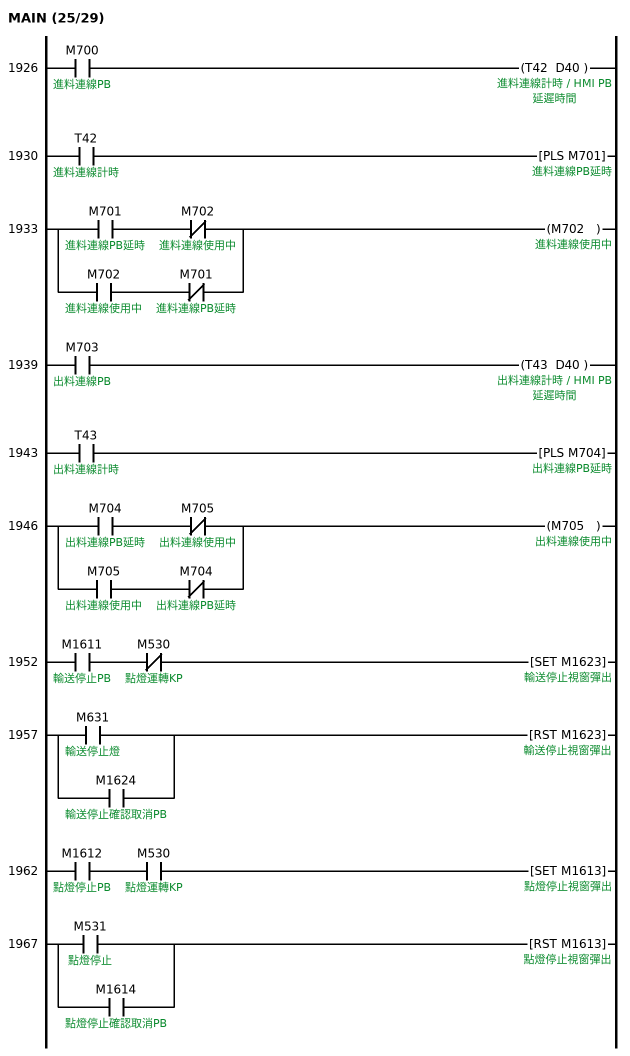
[picture p24: ladder of MAIN, rungs at steps 1926 to 1967]
1926  LD      M700  ; 進料連線PB
      OUT     T42 D40  ; 進料連線計時 / HMI PB  延遲時間
1930  LD      T42  ; 進料連線計時
      PLS     M701  ; 進料連線PB延時
1933  LD      M701  ; 進料連線PB延時
      ANI     M702  ; 進料連線使用中
      LD      M702  ; 進料連線使用中
      ANI     M701  ; 進料連線PB延時
      ORB
      OUT     M702  ; 進料連線使用中
1939  LD      M703  ; 出料連線PB
      OUT     T43 D40  ; 出料連線計時 / HMI PB  延遲時間
1943  LD      T43  ; 出料連線計時
      PLS     M704  ; 出料連線PB延時
1946  LD      M704  ; 出料連線PB延時
      ANI     M705  ; 出料連線使用中
      LD      M705  ; 出料連線使用中
      ANI     M704  ; 出料連線PB延時
      ORB
      OUT     M705  ; 出料連線使用中
1952  LD      M1611  ; 輸送停止PB
      ANI     M530  ; 點燈運轉KP
      SET     M1623  ; 輸送停止視窗彈出
1957  LD      M631  ; 輸送停止燈
      OR      M1624  ; 輸送停止確認取消PB
      RST     M1623  ; 輸送停止視窗彈出
1962  LD      M1612  ; 點燈停止PB
      AND     M530  ; 點燈運轉KP
      SET     M1613  ; 點燈停止視窗彈出
1967  LD      M531  ; 點燈停止
      OR      M1614  ; 點燈停止確認取消PB
      RST     M1613  ; 點燈停止視窗彈出
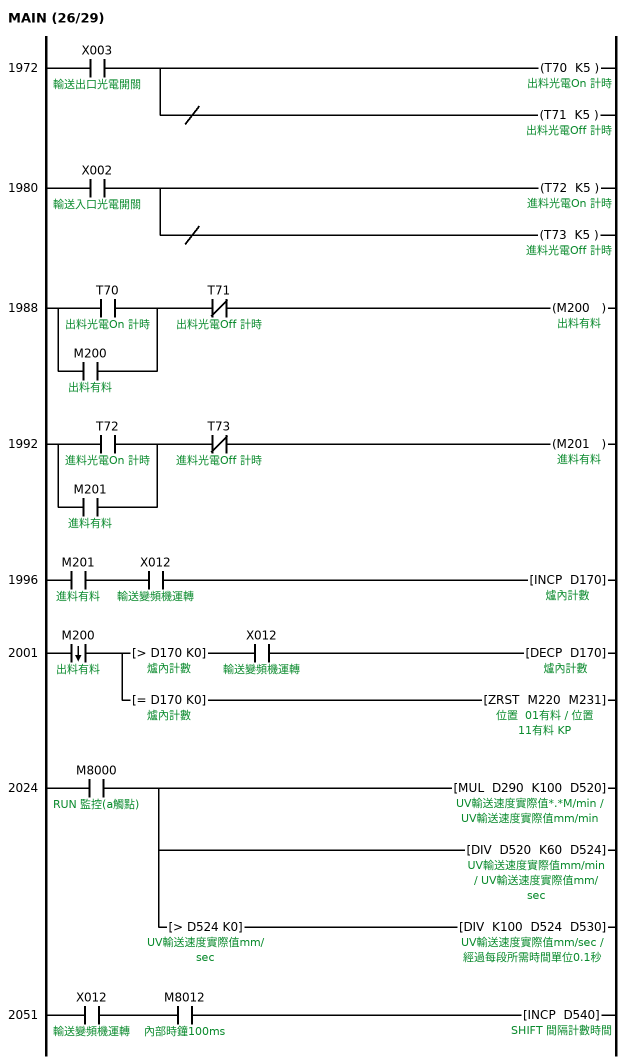
1972  LD      X003  ; 輸送出口光電開關
      OUT     T70 K5  ; 出料光電On 計時
      INV
      OUT     T71 K5  ; 出料光電Off 計時
1980  LD      X002  ; 輸送入口光電開關
      OUT     T72 K5  ; 進料光電On 計時
      INV
      OUT     T73 K5  ; 進料光電Off 計時
1988  LD      T70  ; 出料光電On 計時
      OR      M200  ; 出料有料
      ANI     T71  ; 出料光電Off 計時
      OUT     M200  ; 出料有料
1992  LD      T72  ; 進料光電On 計時
      OR      M201  ; 進料有料
      ANI     T73  ; 進料光電Off 計時
      OUT     M201  ; 進料有料
1996  LD      M201  ; 進料有料
      AND     X012  ; 輸送變頻機運轉
      INCP    D170
2001  LDF     M200  ; 出料有料
      MPS
      AND>    D170 K0  ; 爐內計數
      AND     X012  ; 輸送變頻機運轉
      DECP    D170
      MPP
      AND=    D170 K0  ; 爐內計數
      ZRST    M220 M231  ; 位置  01有料 / 位置  11有料 KP
2024  LD      M8000  ; RUN 監控(a觸點)
      MUL     D290 K100 D520  ; UV輸送速度實際值mm/min
      DIV     D520 K60 D524  ; UV輸送速度實際值mm/sec
      AND>    D524 K0  ; UV輸送速度實際值mm/sec
      DIV     K100 D524 D530  ; 經過每段所需時間單位0.1秒
2051  LD      X012  ; 輸送變頻機運轉
      AND     M8012  ; 內部時鐘100ms
      INCP    D540  ; SHIFT 間隔計數時間
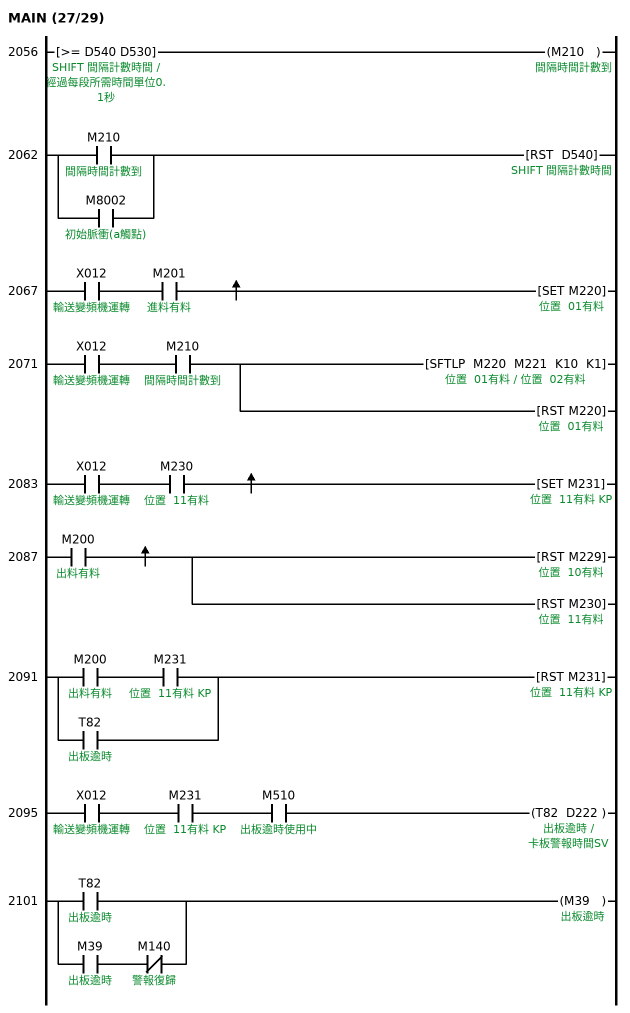
2056  LD>=    D540 D530  ; SHIFT 間隔計數時間 / 經過每段所需時間單位0.1秒
      OUT     M210  ; 間隔時間計數到
2062  LD      M210  ; 間隔時間計數到
      OR      M8002  ; 初始脈衝(a觸點)
      RST     D540  ; SHIFT 間隔計數時間
2067  LD      X012  ; 輸送變頻機運轉
      AND     M201  ; 進料有料
      MEP
      SET     M220  ; 位置  01有料
2071  LD      X012  ; 輸送變頻機運轉
      AND     M210  ; 間隔時間計數到
      SFTLP   M220 M221 K10 K1  ; 位置  02有料
      RST     M220  ; 位置  01有料
2083  LD      X012  ; 輸送變頻機運轉
      AND     M230  ; 位置  11有料
      MEP
      SET     M231  ; 位置  11有料 KP
2087  LD      M200  ; 出料有料
      MEP
      RST     M229  ; 位置  10有料
      RST     M230  ; 位置  11有料
2091  LD      M200  ; 出料有料
      AND     M231  ; 位置  11有料 KP
      OR      T82  ; 出板逾時
      RST     M231  ; 位置  11有料 KP
2095  LD      X012  ; 輸送變頻機運轉
      AND     M231  ; 位置  11有料 KP
      AND     M510  ; 出板逾時使用中
      OUT     T82 D222  ; 出板逾時 / 卡板警報時間SV
2101  LD      T82  ; 出板逾時
      LD      M39  ; 出板逾時
      ANI     M140  ; 警報復歸
      ORB
      OUT     M39  ; 出板逾時
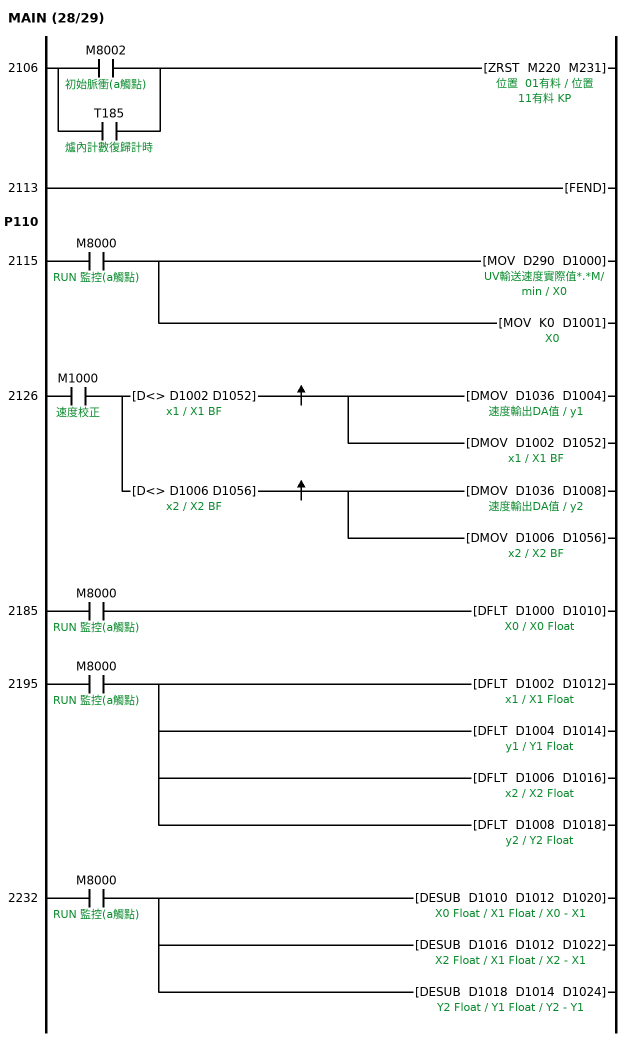
2106  LD      M8002  ; 初始脈衝(a觸點)
      OR      T185  ; 爐內計數復歸計時
      ZRST    M220 M231
2113  FEND
      P110
2115  LD      M8000  ; RUN 監控(a觸點)
      MOV     D290 D1000  ; X0
      MOV     K0 D1001  ; X0
2126  LD      M1000  ; 速度校正
      MPS
      ANDD<>  D1002 D1052  ; x1 / X1 BF
      MEP
      DMOV    D1036 D1004  ; y1
      DMOV    D1002 D1052
      MPP
      ANDD<>  D1006 D1056  ; x2 / X2 BF
      MEP
      DMOV    D1036 D1008  ; y2
      DMOV    D1006 D1056
2185  LD      M8000  ; RUN 監控(a觸點)
      DFLT    D1000 D1010  ; X0 Float
2195  LD      M8000  ; RUN 監控(a觸點)
      DFLT    D1002 D1012  ; X1 Float
      DFLT    D1004 D1014  ; Y1 Float
      DFLT    D1006 D1016  ; X2 Float
      DFLT    D1008 D1018  ; Y2 Float
2232  LD      M8000  ; RUN 監控(a觸點)
      DESUB   D1010 D1012 D1020  ; X0 - X1
      DESUB   D1016 D1012 D1022  ; X2 - X1
      DESUB   D1018 D1014 D1024  ; Y2 - Y1
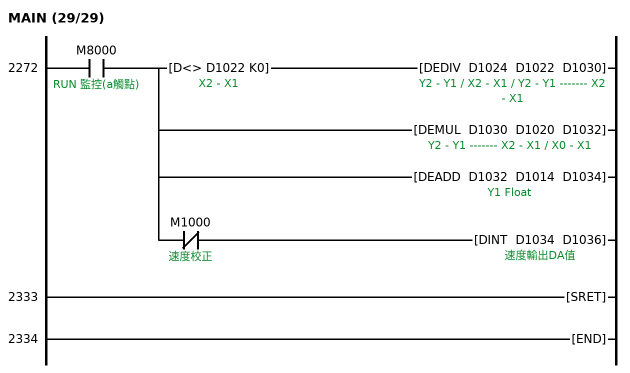
2272  LD      M8000  ; RUN 監控(a觸點)
      MPS
      ANDD<>  D1022 K0  ; X2 - X1
      DEDIV   D1024 D1022 D1030  ; Y2 - Y1 ------- X2 - X1
      MPP
      DEMUL   D1030 D1020 D1032
      DEADD   D1032 D1014 D1034
      ANI     M1000  ; 速度校正
      DINT    D1034 D1036
2333  SRET
2334  END
END_PROGRAM

// device comments not shown above
X030  ; 排風溫度異常
Y025  ; 第 2 燈管啟動信號
M222  ; 位置  03有料
M223  ; 位置  04有料
M224  ; 位置  05有料
M225  ; 位置  06有料
M226  ; 位置  07有料
M227  ; 位置  08有料
M228  ; 位置  09有料
M403  ; UV4自動點燈
M404  ; UV5自動點燈
M405  ; UV6自動點燈
M412  ; UV 3    自動熄燈
M414  ; UV5自動熄燈
M415  ; UV6自動熄燈
M506  ; 省電模式PB
M508  ; 省電模式PLS
M521  ; 出口計數
M598  ; 使用時間歸零PB  (下燈3)
M599  ; 使用時間歸零PB  (上燈3)
M621  ; 下燈3點燈 選擇PB
M622  ; 上燈3點燈 選擇PB
M1246  ; 交握測試PB
M1247  ; 交握測試PB
M1950  ; 上游交握重置PB
M1951  ; 下游交握重置PB
M1960  ; 上游交握重置
M1961  ; 下游交握重置
M2100  ; 物件流入
M2101  ; 接收完成無異常
M2200  ; 開機運轉中-->上游
M2201  ; 允許進料-->上游
M2202  ; 接收完成-->上游
M2204  ; 允許進料保持
M2209  ; IN OVER
M2210  ; 開機運轉中-->下游
M2211  ; 出料請求-->下游
M2212  ; 出料中-->下游
M2219  ; OUT OVER
M2230  ; 出口光電開關
M2301  ; Tact Time保持
M3000  ; 程式目錄
M3001  ; UV燈
M3002  ; UV燈使用時間
M3003  ; 輸送/風車
M3004  ; 速度產量
M3005  ; FX3G-1DA輸出模組
M3006  ; 異常信號
M3007  ; FX2N-2LC溫度
M3008  ; 保養提示
M6105  ; 下游交渥中
M6106  ; 上游-->出料請求ON
T34  ; 省電模式計時
T193  ; 出口光電Off 計時
D160  ; 爐內限制片數SV
D1098  ; 萬用密碼
D1320  ; T0時間設定
D1322  ; T1時間設定
D1323  ; T2時間設定
D1324  ; T3時間設定
D1325  ; T4時間設定
D6000  ; T0時間
D6001  ; T1時間
D6002  ; T3時間
D6004  ; T2時間
D6005  ; T4時間
